INTERFACE I_MotionAxisReset

END_INTERFACE

(* stored: Version 1.1.0.1
   Itf I_MotionAxisReset: Id {fd2e2915-3df3-4ed0-bc4e-9cbc72f9a78c} *)
